// TIA Portal V20 export
FUNCTION_BLOCK "LER_EQP_Interface_Inspection"   // FB127, LAD
// stored: Access Published, MemoryReserve 100, SetENOAutomatically false
   VAR_INPUT
      enable : Bool;
      executeCmd : Bool;
      clock : Bool;
      heartBeat : Byte;
      unitStatus : "LAF_typeUnitStatus";
      unitAlarms : "LAF_typeAlarms";
   END_VAR
   VAR_OUTPUT
      error : Bool;
      status : Word;
   END_VAR
   VAR_IN_OUT
      inspectionCommunication : "LER_typeCommunicationInspection";
      configuration : "LER_typeCommunicationConfiguration";
      moduleInterface : "LER_typeCommunicationInterface";
      controlNode : "LER_typeCommunicationControlNode";
   END_VAR
   VAR
      instEQP_Interface_Communication { S7_SetPoint := 'True'} : "LER_EQP_Communication";
      statInsHeartBeat : Byte;
      statStackState : Struct
         Stop : Bool;
         Abort : Bool;
         Hold : Bool;
         Complete : Bool;
         Idle : Bool;
         TotalStop : Bool;
      END_STRUCT;
      statTonTimer : Array[0..9] of TON_TIME;
      statTofTimer : Array[0..9] of TOF_TIME;
   END_VAR
   VAR CONSTANT
      STATUS_NO_ERROR_OCCURRED : Word := 16#0;
      ERR_HEARTBEAT_ERROR : Word := 16#8000;
   END_VAR
BEGIN

REGION Network 1: EQP Interface Stack State
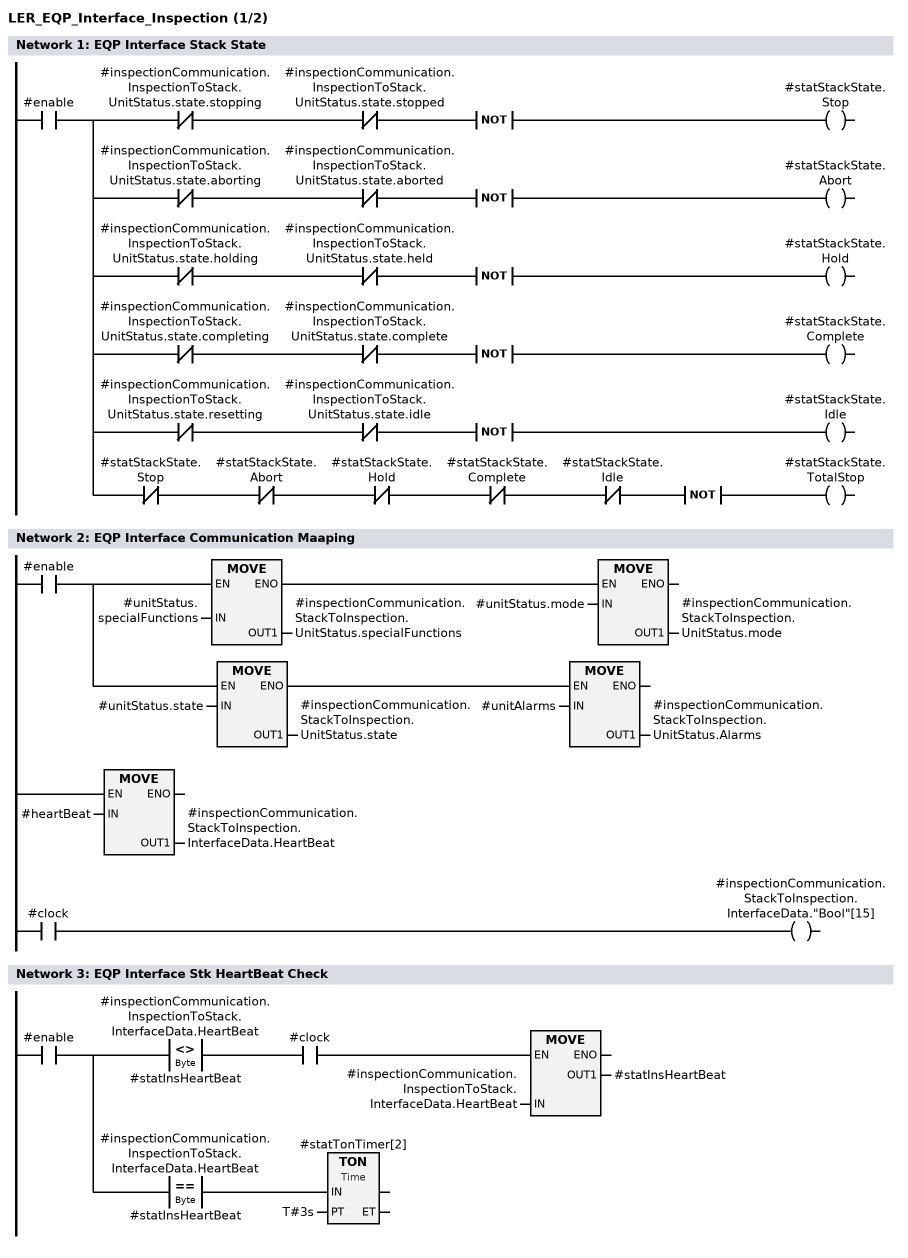
   RUNG wire#powerrail
      Contact( #enable )
      wire#w1
      I_Contact( #inspectionCommunication.InspectionToStack.UnitStatus.state.stopping )
      I_Contact( #inspectionCommunication.InspectionToStack.UnitStatus.state.stopped )
      Not()
      Coil( #statStackState.Stop )
   END_RUNG
   RUNG wire#w1
      I_Contact( #inspectionCommunication.InspectionToStack.UnitStatus.state.aborting )
      I_Contact( #inspectionCommunication.InspectionToStack.UnitStatus.state.aborted )
      Not()
      Coil( #statStackState.Abort )
   END_RUNG
   RUNG wire#w1
      I_Contact( #inspectionCommunication.InspectionToStack.UnitStatus.state.holding )
      I_Contact( #inspectionCommunication.InspectionToStack.UnitStatus.state.held )
      Not()
      Coil( #statStackState.Hold )
   END_RUNG
   RUNG wire#w1
      I_Contact( #inspectionCommunication.InspectionToStack.UnitStatus.state.completing )
      I_Contact( #inspectionCommunication.InspectionToStack.UnitStatus.state.complete )
      Not()
      Coil( #statStackState.Complete )
   END_RUNG
   RUNG wire#w1
      I_Contact( #inspectionCommunication.InspectionToStack.UnitStatus.state.resetting )
      I_Contact( #inspectionCommunication.InspectionToStack.UnitStatus.state.idle )
      Not()
      Coil( #statStackState.Idle )
   END_RUNG
   RUNG wire#w1
      I_Contact( #statStackState.Stop )
      I_Contact( #statStackState.Abort )
      I_Contact( #statStackState.Hold )
      I_Contact( #statStackState.Complete )
      I_Contact( #statStackState.Idle )
      Not()
      Coil( #statStackState.TotalStop )
   END_RUNG
   // the same network as SCL:
   #statStackState.Stop := NOT (#enable AND NOT #inspectionCommunication.InspectionToStack.UnitStatus.state.stopping AND NOT #inspectionCommunication.InspectionToStack.UnitStatus.state.stopped);
   #statStackState.Abort := NOT (#enable AND NOT #inspectionCommunication.InspectionToStack.UnitStatus.state.aborting AND NOT #inspectionCommunication.InspectionToStack.UnitStatus.state.aborted);
   #statStackState.Hold := NOT (#enable AND NOT #inspectionCommunication.InspectionToStack.UnitStatus.state.holding AND NOT #inspectionCommunication.InspectionToStack.UnitStatus.state.held);
   #statStackState.Complete := NOT (#enable AND NOT #inspectionCommunication.InspectionToStack.UnitStatus.state.completing AND NOT #inspectionCommunication.InspectionToStack.UnitStatus.state.complete);
   #statStackState.Idle := NOT (#enable AND NOT #inspectionCommunication.InspectionToStack.UnitStatus.state.resetting AND NOT #inspectionCommunication.InspectionToStack.UnitStatus.state.idle);
   #statStackState.TotalStop := NOT (#enable AND NOT #statStackState.Stop AND NOT #statStackState.Abort AND NOT #statStackState.Hold AND NOT #statStackState.Complete AND NOT #statStackState.Idle);
END_REGION

REGION Network 2: EQP Interface Communication Maaping
   RUNG wire#powerrail
      Contact( #enable )
      wire#w1
      Move(in := #unitStatus.specialFunctions, out1 => #inspectionCommunication.StackToInspection.UnitStatus.specialFunctions)
      Move(in := #unitStatus.mode, out1 => #inspectionCommunication.StackToInspection.UnitStatus.mode)
   END_RUNG
   RUNG wire#w1
      Move(in := #unitStatus.state, out1 => #inspectionCommunication.StackToInspection.UnitStatus.state)
      Move(in := #unitAlarms, out1 => #inspectionCommunication.StackToInspection.UnitStatus.Alarms)
   END_RUNG
   RUNG wire#powerrail
      Move(in := #heartBeat, out1 => #inspectionCommunication.StackToInspection.InterfaceData.HeartBeat)
   END_RUNG
   RUNG wire#powerrail
      Contact( #clock )
      Coil( #inspectionCommunication.StackToInspection.InterfaceData."Bool"[15] )
   END_RUNG
   // the same network as SCL:
   IF #enable THEN
       #inspectionCommunication.StackToInspection.UnitStatus.specialFunctions := #unitStatus.specialFunctions;
       #inspectionCommunication.StackToInspection.UnitStatus.mode := #unitStatus.mode;
       #inspectionCommunication.StackToInspection.UnitStatus.state := #unitStatus.state;
       #inspectionCommunication.StackToInspection.UnitStatus.Alarms := #unitAlarms;
   END_IF;
   #inspectionCommunication.StackToInspection.InterfaceData.HeartBeat := #heartBeat;
   #inspectionCommunication.StackToInspection.InterfaceData."Bool"[15] := #clock;
END_REGION

REGION Network 3: EQP Interface Stk HeartBeat Check
   RUNG wire#powerrail
      Contact( #enable )
      wire#w1
      { S7_Templates := "SrcType := Byte" } NE_Contact(in1 := #inspectionCommunication.InspectionToStack.InterfaceData.HeartBeat, in2 := #statInsHeartBeat)
      Contact( #clock )
      Move(in := #inspectionCommunication.InspectionToStack.InterfaceData.HeartBeat, out1 => #statInsHeartBeat)
   END_RUNG
   RUNG wire#w1
      { S7_Templates := "SrcType := Byte" } EQ_Contact(in1 := #inspectionCommunication.InspectionToStack.InterfaceData.HeartBeat, in2 := #statInsHeartBeat)
      { S7_Templates := "time_type := Time" } #statTonTimer[2].TON(pt := T#3s, et =>)
   END_RUNG
   // the same network as SCL:
   IF #enable AND (#inspectionCommunication.InspectionToStack.InterfaceData.HeartBeat <> #statInsHeartBeat) AND #clock THEN
       #statInsHeartBeat := #inspectionCommunication.InspectionToStack.InterfaceData.HeartBeat;
   END_IF;
   #statTonTimer[2].TON(IN := #enable AND (#inspectionCommunication.InspectionToStack.InterfaceData.HeartBeat = #statInsHeartBeat),
                        PT := T#3s);
END_REGION

REGION Network 4: EQP Interface Communication Stack <-> ReelCut
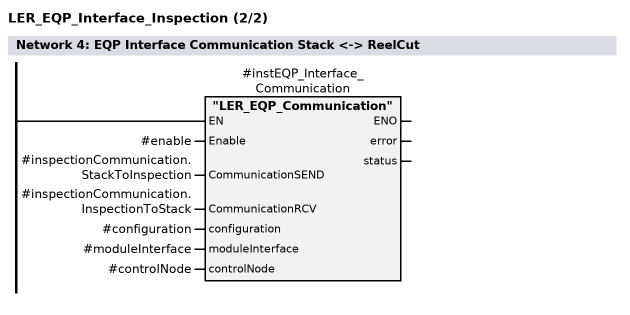
   RUNG wire#powerrail
      #instEQP_Interface_Communication(Enable := #enable, CommunicationSEND := #inspectionCommunication.StackToInspection, CommunicationRCV := #inspectionCommunication.InspectionToStack, configuration := #configuration, moduleInterface := #moduleInterface, controlNode := #controlNode, error =>, status =>)
   END_RUNG
   // the same network as SCL:
   #instEQP_Interface_Communication(Enable := #enable,   // "LER_EQP_Communication"
                           CommunicationSEND := #inspectionCommunication.StackToInspection,
                           CommunicationRCV := #inspectionCommunication.InspectionToStack,
                           configuration := #configuration,
                           moduleInterface := #moduleInterface,
                           controlNode := #controlNode);
END_REGION

REGION Network 5 (SCL): Error Check
   REGION Error Code Search

       IF #enable AND NOT #configuration.disableAlarms THEN
           IF #statTonTimer[2].Q THEN
               #status := #ERR_HEARTBEAT_ERROR;

           ELSIF #instEQP_Interface_Communication.error THEN
               #status := #instEQP_Interface_Communication.status;

           ELSE
               #status := #STATUS_NO_ERROR_OCCURRED;

           END_IF;
       ELSE
           #status := #STATUS_NO_ERROR_OCCURRED;

       END_IF;


       // Error Bit
       #error := #status <> 0;

   END_REGION
END_REGION

REGION Network 6 (SCL): ##### Outputs mapping #####
   #moduleInterface.monitoring.error := #error;
   #moduleInterface.monitoring.status := #status;

   #controlNode.monitoring := #moduleInterface.monitoring;
END_REGION
END_FUNCTION_BLOCK
